// TIA Portal V17 export
// export: Created 2023-09-10T16:27:52.6737566Z, ExportSetting WithDefaults, DisplayName Totally Integrated Automation Portal, DisplayVersion V17, DisplayName TIA Portal Openness, DisplayVersion V17, DisplayName TIA Portal Version Control Interface, DisplayVersion V17, DisplayName STEP 7 Professional, DisplayVersion V17, DisplayName STEP 7 Safety, DisplayVersion V17, DisplayName WinCC Advanced, DisplayVersion V17
DATA_BLOCK "modbus"   // DB3
{ S7_Optimized_Access := 'FALSE'; DB_Accessible_From_OPC_UA := 'FALSE' }
VERSION : 0.1
// stored: AutoNumber true, DBAccessibleFromOPCUA false, IsOnlyStoredInLoadMemory false, IsWriteProtectedInAS false
   VAR
      rs485parity : Int := 0;
      rs485baudrate : Int := 9600;
      modbusEncoderAdd : Int := 1;
      modbusMode : Int := 0;
      modbusEncoderDataRegister : DInt := 40001;
      modbusDataLength : DInt := 1;
      encoderMaxValue : DInt := 1024;
      mbLoadError : Bool;
      mbLoadDone : Bool;
      mbLoadStatus : Word;
      mbMasterBusy : Bool;
      mbMasterDone : Bool;
      mbMasterError : Bool;
      mbMasterStatus : Word;
      modbusReqBit : Bool;
      modbusReqAgainBit : Bool;
      modbusTimer : IEC_TIMER;
      REGISTERS : Array[0..9] of Int;
      lastEncoderValue : Int;
   END_VAR
BEGIN
   modbusTimer.PT := T#2S;
END_DATA_BLOCK
